// TIA Portal V20 export
DATA_BLOCK "F-link_DB"   // DB2
{ S7_Optimized_Access := 'TRUE' }
// stored: MemoryReserve 100
   VAR
      receive : "F-link_UDT";
   END_VAR
BEGIN
END_DATA_BLOCK
